(* IEC 61131-3 sources: eCockpitGit/test_project/src/%PLC%PLCTest2/%PLOG%Plc Logic/%APP%APP1_Test/%POU%prg_test, 1 file *)

(* ---- %METH%METHy.st ---- *)
METHOD METHy : BOOL
VAR_INPUT
END_VAR

(*%!%__DELIMITER__%!%*)
